# EPICS autosave request: iocs/ADCrayDlIOC/iocBoot/iocHDF5Test/auto_settings.req
file "CrayDl_settings.req",    P=$(P),  R=cam1:
file "CrayDl_settings.req",    P=$(P),  R=cam2:
file "NDStdArrays_settings.req",    P=$(P),  R=image1:
file "commonPlugin_settings.req",   P=$(P)
